FUNCTION_BLOCK INTERNAL FB_LightTowerComponent_Tests EXTENDS FB_TestSuite
VAR_INPUT
END_VAR
VAR_OUTPUT
END_VAR
VAR
	componentItem	: BOOL;
END_VAR

Test01_AllFunctionalityTests();

METHOD Test01_AllFunctionalityTests 
VAR_INST
	timer	 		: Tc2_Standard.TON;
	timerOff		: Tc2_Standard.TON;
	component		: FB_LightTowerComponent := (component := componentItem);
	onOffTestDone	: BOOL;
END_VAR
IF TcUnit.TEST_ORDERED('Test01_AllFunctionalityTests') THEN
	component();
	IF NOT onOffTestDone THEN
		component.Activate();
		AssertTrue(Condition := component.Value, Message := 'Calling .Activate() should set the .Value property to TRUE.');
		AssertTrue(Condition := componentItem, Message := 'Calling .Activate() should set the referenced variable to TRUE.');
		component.Deactivate();
		AssertFalse(Condition := component.Value, Message := 'Calling .Deactivate() should set the .Value property to FALSE.');
		AssertFalse(Condition := componentItem, Message := 'Calling .Deactivate() should set the referenced variable to FALSE.');
		onOffTestDone := TRUE;
	END_IF
	
	component.PulseWithInterval(DurationOn := T#100MS, DurationOff := T#100MS);
	timer(in := TRUE, PT := T#100MS);
	IF NOT timer.Q THEN
		AssertTrue(Condition := component.Value, Message := 'Component.Value should be TRUE until duration on is elapsed.');
		AssertTrue(Condition := componentItem, Message := 'Referenced variable should be TRUE until duration on is elapsed.');
	ELSE
		timerOff(IN := TRUE, PT := T#100MS);
		IF timerOff.Q THEN
			AssertTrue(Condition := component.Value, Message := 'Component.Value should be TRUE when duration off is elapsed.');
			AssertTrue(Condition := componentItem, Message := 'Reference variable should be TRUE when duration off is elapsed.');
			TcUnit.TEST_FINISHED();
			RETURN;
		END_IF
		AssertFalse(Condition := component.Value, Message := 'Component.Value should be FALSE until duration off is elapsed.');
		AssertFalse(Condition := componentItem, Message := 'Reference variable should be FALSE until duration off is elapsed.');
	END_IF	
END_IF
END_METHOD

END_FUNCTION_BLOCK

(* stored: Version 1.1.0.1, ProductVersion 3.1.4024.16
   POU FB_LightTowerComponent_Tests: Id {d730fdac-a82d-014c-34ad-463aa6395209}, SpecialFunc None
   Method Test01_AllFunctionalityTests: Id {a0beeec2-3445-0515-3ad9-48d21260790b} *)
